INTERFACE I_TraceSourceInfo EXTENDS I_Base

{attribute 'monitoring':='call'}
PROPERTY SourceId : UDINT
GET
END_GET
END_PROPERTY

{attribute 'monitoring':='call'}
PROPERTY SourceName : T_MaxString
GET
END_GET
END_PROPERTY

{attribute 'monitoring':='call'}
PROPERTY TimeStamp : ULINT
GET
END_GET
END_PROPERTY

END_INTERFACE

(* stored: Version 1.1.0.1, ProductVersion 3.1.4026.18
   Itf I_TraceSourceInfo: Id {88aae583-53c4-086d-17ad-e3f03a973024}
   Property SourceId: Id {f63793bb-f5e5-09f5-30e8-57e18b6bba04}
   Get Get: Id {4e0c3652-ce73-01bd-153d-bf5fdfc22e92}
   Property SourceName: Id {502eeb65-2317-0609-2ba6-57ba9b293fb2}
   Get Get: Id {a77f477b-ecc3-0391-16c6-dc678118aa4b}
   Property TimeStamp: Id {2adcebfe-6e29-0498-0ede-1e0e37c5f0a7}
   Get Get: Id {3612711f-962a-0d9e-3258-1dd00344b42f} *)
